FUNCTION FC1_Bereken_Snelheid : DINT
VAR_INPUT
    Laadgewicht : DINT;    // Invoer van de weegcel
    MinLaad     : DINT;    // Minimum laadgewicht (lege transportband)
    MaxLaad     : DINT;    // Maximum laadgewicht (volgeladen transportband)
    MinSnelheid : REAL;    // Minimum transportbandsnelheid (langzaamst)
    MaxSnelheid : REAL;    // Maximum transportbandsnelheid (snelst)
END_VAR

VAR
    LaadRatio   : DINT;    	// Proportionele waarde van het laadgewicht
	LaadRatioReal : REAL;	// vertaald naar REAL
    BerekendeSnelheid : REAL; // De berekende snelheid in REAL
END_VAR



// Zorg ervoor dat Laadgewicht binnen de grenzen valt
IF Laadgewicht < MinLaad THEN
    Laadgewicht := MinLaad + 2 ;
ELSIF Laadgewicht > MaxLaad THEN
    Laadgewicht := MaxLaad;
END_IF

// Bereken de laadratio als percentage van het maximale laadgewicht
LaadRatio := (Laadgewicht - MinLaad) / (MaxLaad - MinLaad);

//conversie naar Real
LaadRatioReal := DINT_TO_REAL(LaadRatio);

// Bereken de transportbandsnelheid op basis van de laadratio
BerekendeSnelheid := MaxSnelheid - (LaadRatioReal * (MaxSnelheid - MinSnelheid));

// Rond de berekende snelheid af naar een DINT waarde en retourneer deze
FC1_Bereken_Snelheid := REAL_TO_DINT(BerekendeSnelheid);

END_FUNCTION

(* stored: Version 1.1.0.1, ProductVersion 3.1.4024.12
   POU FC1_Bereken_Snelheid: Id {12de46b1-cd22-4bee-b0d4-4edb4530f63f}, SpecialFunc None *)
